(* Schneider Machine Expert - Basic project Multi POU template, file version 3.0.0.0 *)
(* ProjectInformations: Name=New project *)

HARDWARE
  Cpu 0: TM221CE16U
  EthernetConfiguration: NetworkName=M221, IpAllocationMode=FixedAddress, IpAddress=0.0.0.0, SubnetMask=0.0.0.0
  SerialLineConfiguration: Baud=Baud19200, Parity=ParityEven, DataBits=DataBits8, StopBits=StopBits1, PhysicalMedium=PhysicalMediumRs485, TransmissionMode=TransmissionModeModbusRtu, SlaveId=1, Addressing=SlaveAddressing
  MastTask: UsePeriodScanMode=false, PeriodScan=100
  FastTask: Period=255
  CpuBehavior: StartingMode=StartAsPreviousState, AutoSaveRamOnEeprom=true, WatchdogPeriod=250

SYMBOLS  (address, symbol, comment, settings)
  %M0       SYS_READY
  %M1       MANUAL_MODE
  %M2       AUTO_MODE
  %S0       SB_COLDSTART  "Indicates or executes a cold start (data initialized to default values)"
  %S1       SB_WARMSTART  "Indicates there was a warm start with data backup"
  %MW10     AUTO_MANUAL_SELECTION
  %TM0        [Preset=3, Base=OneSecond]
  %I0.0     EMERGENCY_PB

POU System_Init
  (* SectionNumber=0 *)

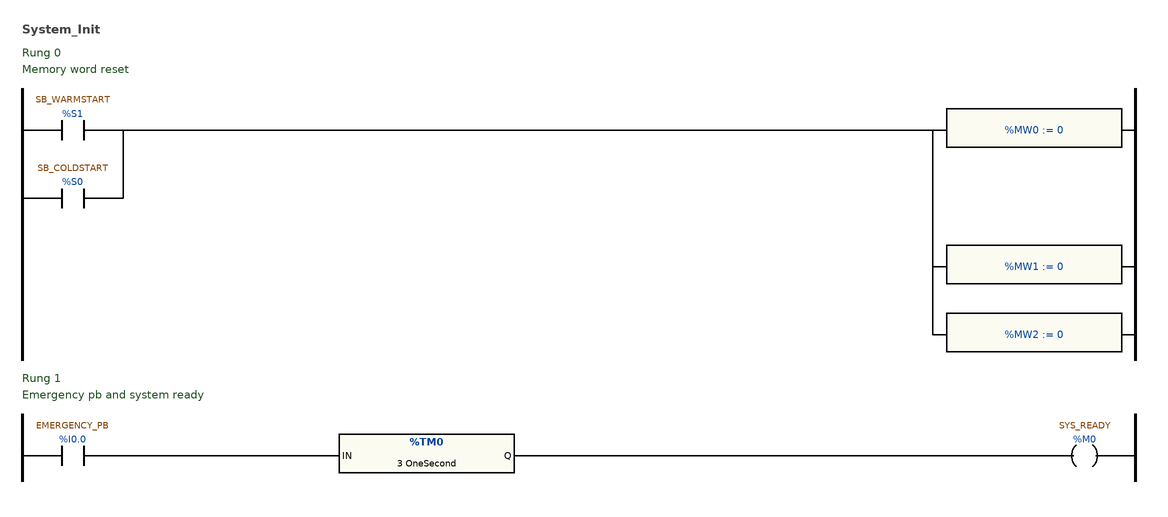

// Rung 0
// Memory word reset
  LD %S1                  (* SB_WARMSTART *)
  OR %S0                  (* SB_COLDSTART *)
  [ %MW0 := 0 ]
  [ %MW1 := 0 ]
  [ %MW2 := 0 ]
  // as ST:
  //   IF SB_WARMSTART OR SB_COLDSTART THEN %MW0 := 0; END_IF;
  //   IF SB_WARMSTART OR SB_COLDSTART THEN %MW1 := 0; END_IF;
  //   IF SB_WARMSTART OR SB_COLDSTART THEN %MW2 := 0; END_IF;

// Rung 1
// Emergency pb and system ready
  BLK %TM0
  LD %I0.0                (* EMERGENCY_PB *)
  IN
  OUT_BLK
  LD Q
  ST %M0                  (* SYS_READY *)
  END_BLK
  // as ST:
  //   %TM0(IN := EMERGENCY_PB);
  //   SYS_READY := %TM0.Q;

POU Manual
  (* SectionNumber=0 *)

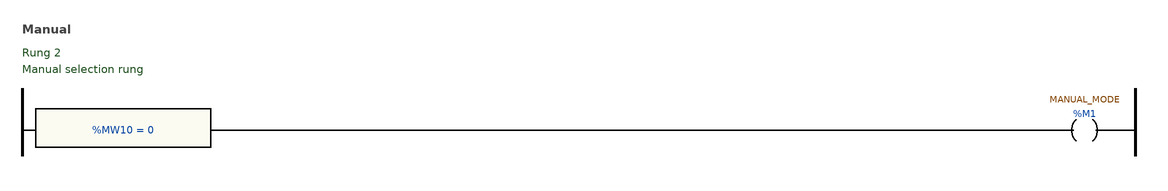

// Rung 2
// Manual selection rung
  LD [ %MW10 = 0 ]        (* AUTO_MANUAL_SELECTION *)
  ST %M1                  (* MANUAL_MODE *)
  // as ST:
  //   MANUAL_MODE := AUTO_MANUAL_SELECTION = 0;

POU Auto
  (* SectionNumber=0 *)

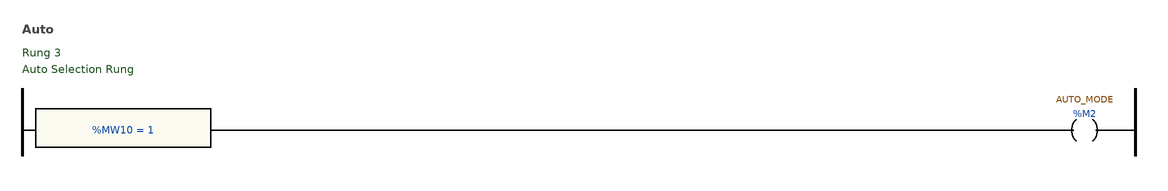

// Rung 3
// Auto Selection Rung
  LD [ %MW10 = 1 ]        (* AUTO_MANUAL_SELECTION *)
  ST %M2                  (* AUTO_MODE *)
  // as ST:
  //   AUTO_MODE := AUTO_MANUAL_SELECTION = 1;
